TYPE DUT_SENSOR_DATAS_6 :
UNION
	data_lreal:REAL;
	data_byte:ARRAY[0..3] OF BYTE;
END_UNION
END_TYPE

(* stored: Version 1.1.0.1, ProductVersion 3.1.4024.6
   DUT DUT_SENSOR_DATAS_6: Id {7722bcd5-6bbf-4a26-94e1-73f625d399a4} *)
